// SIMATIC STEP 7 (V5.x) project ZEn01_09_STEP7__Zebra
// CPU: CPU314(1)
// station: Hardware
// station: SIMATIC 300(1)
// program: S7-Program(1)

SYMBOL_TABLE
"Switch_right"	I 0.0	BOOL	// Switch on the right side of the street
"Switch_left"	I 0.1	BOOL	// Switch on the left side of the street
"Pedestrian_light"	M 0.0	BOOL	// Memory bit for switching traffic light on request for green by a pedestrian
"Ped_red"	Q 0.0	BOOL	// Red for pedestrians
"Ped_green"	Q 0.1	BOOL	// Green for pedestrians
"Car_red"	Q 0.5	BOOL	// Red for cars
"Car_orange"	Q 0.6	BOOL	// Orange for cars
"Car_green"	Q 0.7	BOOL	// Green for cars
"Car_orange_phase"	T 2	TIMER	// Duration of orange phase for cars
"Ped_green_phase"	T 3	TIMER	// Duration of green phase for pedestrians
"Car_delay_red"	T 4	TIMER	// Delay red phase for cars
"Car_red_orange_phase"	T 5	TIMER	// Duration of red/orange phase for cars
"Ped_delay_green"	T 6	TIMER	// Delay next green request for pedestrians
END_SYMBOL_TABLE

FUNCTION FC 1 : VOID
TITLE = Sample program TRAFFIC LIGHT
//Control for a pedestrian crosswalk traffic light
//
VERSION : 0.0
BEGIN
NETWORK
TITLE = Determining green request for pedestrians
//Determining whether I 0.0 or I 0.1 is set  
      A(;
      A(;
      O     "Switch_right";
      O     "Switch_left";
      );
      A     "Ped_delay_green";
      O     "Pedestrian_light";
      );
      AN    "Car_red_orange_phase";
      =     "Pedestrian_light";
NETWORK
TITLE = Green phase for cars
//If I 0.0 or I 0.1 are not set, the light stays green for cars      
      AN    "Pedestrian_light";
      =     "Car_green";
NETWORK
TITLE = Start timer for orange phase for cars
//If a request for "pedestrian green" is present, the orange phase for cars 
//is started      
      A     "Pedestrian_light";
      L     S5T#3S;
      SD    "Car_orange_phase";
NETWORK
TITLE = Orange phase for cars
//The output Car_orange is activated if a "pedestrian green" 
//is present or at the end of the pedestrian green phase
//and when the red delay for cars has elapsed       
      A     "Pedestrian_light";
      A(;
      ON    "Car_orange_phase";
      O     "Car_delay_red";
      );
      =     "Car_orange";
NETWORK
TITLE = Red phase for cars
//The red phase for cars starts when the "pedestrian green" request 
//is received and when the orange phase for cars has elapsed 
      A     "Pedestrian_light";
      A     "Car_orange_phase";
      =     "Car_red";
NETWORK
TITLE = Start timer for pedestrian green phase
//When the red phase for cars is reached, the green phase for pedestrians
//is started      
      A     "Car_red";
      L     S5T#10S;
      SD    "Ped_green_phase";
NETWORK
TITLE = Green phase for pedestrians
//The pedestrian light remains green for as long as the red phase for cars 
//AND as long as the set time for "pedestrian green" has not elapsed      
      A     "Car_red";
      AN    "Ped_green_phase";
      =     "Ped_green";
NETWORK
TITLE = Start timer for orange phase delay for cars
//When the "pedestrian green" phase has elapsed, the introduction of the
//red/orange phase for cars is delayed      
      A     "Pedestrian_light";
      A     "Ped_green_phase";
      L     S5T#6S;
      SD    "Car_delay_red";
NETWORK
TITLE = Red phase for pedestrians
//The red condition for pedestrians is fulfilled when
//no "pedestrian green" request is present OR 
//a "pedestrian green" request is present AND
//                the green phase for pedestrians has elapsed OR
//                the orange phase for cars has not elapsed      
      A     "Pedestrian_light";
      A(;
      ON    "Car_orange_phase";
      O     "Ped_green_phase";
      );
      ON    "Pedestrian_light";
      =     "Ped_red";
NETWORK
TITLE = Start timer for red/orange phase for cars
//The red/orange phase for cars starts when the delay following the switch
//of the pedestrian light from green to red has elapsed      
      A     "Pedestrian_light";
      A     "Car_delay_red";
      L     S5T#3S;
      SD    "Car_red_orange_phase";
NETWORK
TITLE = Start timer for green request delay
//A new "pedestrian green" request is only possible once the delay time
//has elapsed      
      A     "Car_green";
      L     S5T#1S;
      SD    "Ped_delay_green";
END_FUNCTION

ORGANIZATION_BLOCK OB 1
VERSION : 0.1
VAR_TEMP
  OB1_EV_CLASS : BYTE ;	//Bits 0-3 = 1 (Coming event), Bits 4-7 = 1 (Event class 1)
  OB1_SCAN_1 : BYTE ;	//1 (Cold restart scan 1 of OB 1), 3 (Scan 2-n of OB 1)
  OB1_PRIORITY : BYTE ;	//1 (Priority of 1 is lowest)
  OB1_OB_NUMBR : BYTE ;	//1 (Organization block 1, OB1)
  OB1_RESERVED_1 : BYTE ;	//Reserved for system
  OB1_RESERVED_2 : BYTE ;	//Reserved for system
  OB1_PREV_CYCLE : INT ;	//Cycle time of previous OB1 scan (milliseconds)
  OB1_MIN_CYCLE : INT ;	//Minimum cycle time of OB1 (milliseconds)
  OB1_MAX_CYCLE : INT ;	//Maximum cycle time of OB1 (milliseconds)
  OB1_DATE_TIME : DATE_AND_TIME ;	//Date and time OB1 started
END_VAR
BEGIN
NETWORK
TITLE = Call FC1 for traffic light control
      CALL  FC 1;
      NOP   0;
END_ORGANIZATION_BLOCK
